FUNCTION_BLOCK Sangre
VAR_INPUT
END_VAR
VAR_OUTPUT
END_VAR
VAR
	VarHumano: Humano;
END_VAR

END_FUNCTION_BLOCK

(* stored: Version 1.1.0.1, ProductVersion 3.1.4024.12
   POU Sangre: Id {6d88db65-9f35-4676-beca-8e0c4ab5fbac}, SpecialFunc None *)
